Universal Robots URScript: rtde_control_loop.script

def unnamed():
  set_standard_analog_input_domain(0, 1)
  set_standard_analog_input_domain(1, 1)
  set_tool_analog_input_domain(0, 1)
  set_tool_analog_input_domain(1, 1)
  set_analog_outputdomain(0, 0)
  set_analog_outputdomain(1, 0)
  set_input_actions_to_default()
  set_tool_communication(False, 115200, 0, 1, 1.5, 3.5)
  set_tool_output_mode(0)
  set_tool_digital_output_mode(0, 1)
  set_tool_digital_output_mode(1, 1)
  set_tool_voltage(0)
  set_safety_mode_transition_hardness(1)
  set_gravity([0.0, 0.0, 9.82])
  set_tcp(p[0.0,0.0,0.0,0.0,0.0,0.0])
  set_payload(0.0)
  global Waypoint_1_p=p[-.189631536923, -.609683881651, .260971148694, -.001221359682, 3.116276528482, .038891915637]
  global Waypoint_1_q=[-1.6006999999999998, -1.7271, -2.2029999999999994, -0.8079999999999998, 1.5951, -0.030999999999999694]
  while (True):
    $ 1 "Robot Program"
    $ 2 "MoveP"
    $ 3 "Waypoint_1"
    movep(Waypoint_1_p, a=1.2, v=0.25, r=0.025)
  end
end
